TYPE DUT_Effect_Monoid :
STRUCT
	Count   : INT := 0;
    Effects : ARRAY[1..20] OF DUT_Effect;
END_STRUCT
END_TYPE

(* stored: Version 1.1.0.1
   DUT DUT_Effect_Monoid: Id {cf594f49-7cae-4edd-9d33-a056d15d4f24} *)
